(* CODESYS project I2C_PCF8574_3.library
   Company: Switcher
   DefaultNamespace: IO
   Version: 1.1.0.0
   Description: Library containing device support for 8574 under Raspberry Pi
   Placeholder: PlaceholderTemplate
   Author: Switcher
   Title: Raspberry I2C PCF8574

Project tree, tasks and I/O mapping:
  libraries: Standard, * (System); IoStandard, * (System); Raspberry Pi Peripherals, * (3S - Smart Software Solutions GmbH)
  function block PCF8574 [ST]: AfterReadInputs, BeforeWriteOutputs
  00000000-0000-0000-0000-000000000000|D:\CoDeSys\LibrariesV3\trunk\Intern\CAA\CAA Template\3.4.0.0 draft\Placeholder.xml
  00000000-0000-0000-0000-000000000000|D:\CoDeSys\LibrariesV3\trunk\Intern\CAA\CAA Template\3.2.0.3 draft\Prefix.pdf
  00000000-0000-0000-0000-000000000000|D:\CoDeSys\LibrariesV3\trunk\Intern\CAA\CAA Template\3.5.2.0 draft\Placeholder.xml
*)

// PCF8574
FUNCTION_BLOCK PCF8574 EXTENDS i2c
VAR_INPUT
	PCFOUT: BYTE;
END_VAR
VAR_OUTPUT
	PCFIN: BYTE;	
END_VAR
VAR
//	aby: ARRAY[0..5] OF BYTE;
END_VAR

SUPER^();

CASE _iState OF
0:
	IF usiAddress = 0 THEN
		usiAddress := 16#38;
	END_IF
	
	IF init() THEN
		_iState := 10;
	END_IF	
	
END_CASE

METHOD AfterReadInputs : INT
VAR
	Buffer : ARRAY[0..3] OF BYTE;
	len: dINT;
END_VAR
SUPER^.AfterReadInputs();


IF _iState = 10 THEN
//	timer();
//	IF timer.Q THEN
//		timer(IN := FALSE);
//		timer(IN := TRUE);
		
//		readregister(0, ADR(aby), 3);
		read(ADR(PCFIN), 1);
//		read8(GR0111);

//		iMX := aby[0];
//		iMY := aby[1];
//		iMZ := aby[2];
		
//	END_IF	
END_IF
END_METHOD

METHOD BeforeWriteOutputs : INT
VAR
END_VAR
SUPER^.BeforeWriteOutputs();

IF _iState = 10 THEN

//	write8(16#00, PCFOUT);
	Write(ADR(PCFOUT), 1);
		
END_IF
END_METHOD

END_FUNCTION_BLOCK
